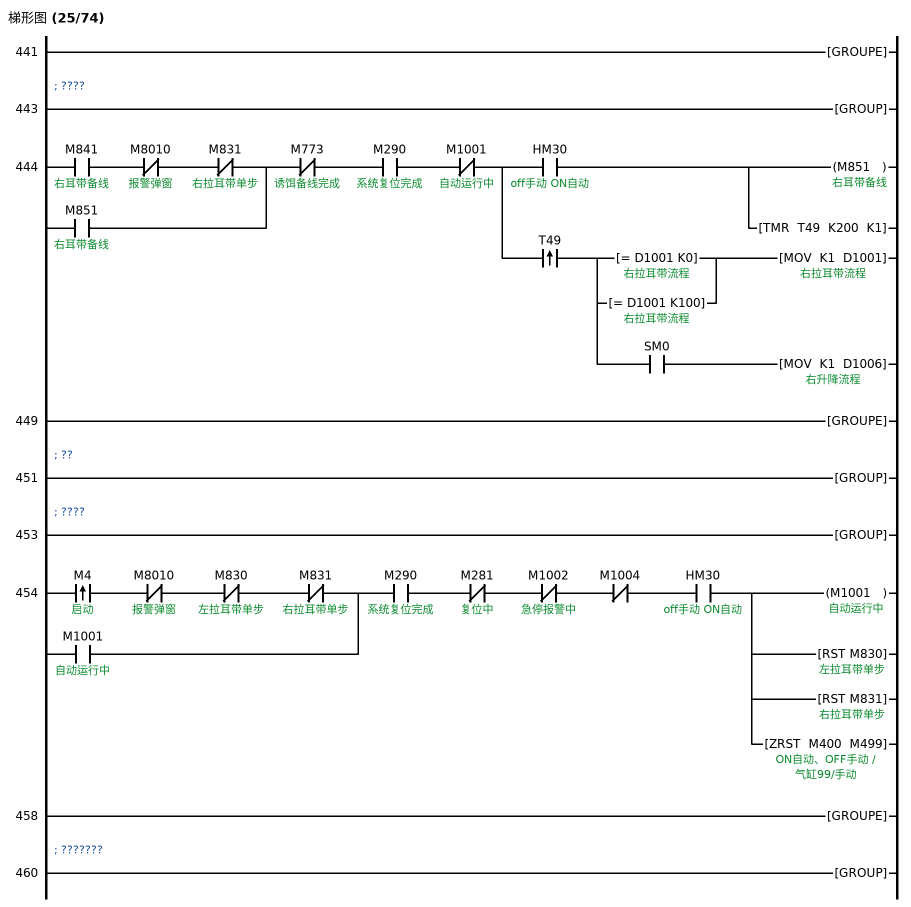
[picture p24: 梯形图 rows 441-460]
GROUPE
; ????
GROUP
LD     M841	; 右耳带备线
ANI    M8010	; 报警弹窗
ANI    M831	; 右拉耳带单步
OR     M851	; 右耳带备线
ANI    M773	; 诱饵备线完成
AND    M290	; 系统复位完成
ANI    M1001	; 自动运行中
MPS
AND    HM30	; off手动 ON自动
OUT    M851	; 右耳带备线
TMR    T49 K200 K1
MPP
ANDP   T49
MPS
LD=    D1001 K0	; 右拉耳带流程
OR=    D1001 K100	; 右拉耳带流程
ANB
MOV    K1 D1001	; 右拉耳带流程
MPP
AND    SM0
MOV    K1 D1006	; 右升降流程
GROUPE
; ??
GROUP
; ????
GROUP
LDP    M4	; 启动
ANI    M8010	; 报警弹窗
ANI    M830	; 左拉耳带单步
ANI    M831	; 右拉耳带单步
OR     M1001	; 自动运行中
AND    M290	; 系统复位完成
ANI    M281	; 复位中
ANI    M1002	; 急停报警中
ANI    M1004
AND    HM30	; off手动 ON自动
OUT    M1001	; 自动运行中
RST    M830	; 左拉耳带单步
RST    M831	; 右拉耳带单步
ZRST   M400 M499	; ON自动、OFF手动 / 气缸99/手动
GROUPE
; ???????
GROUP

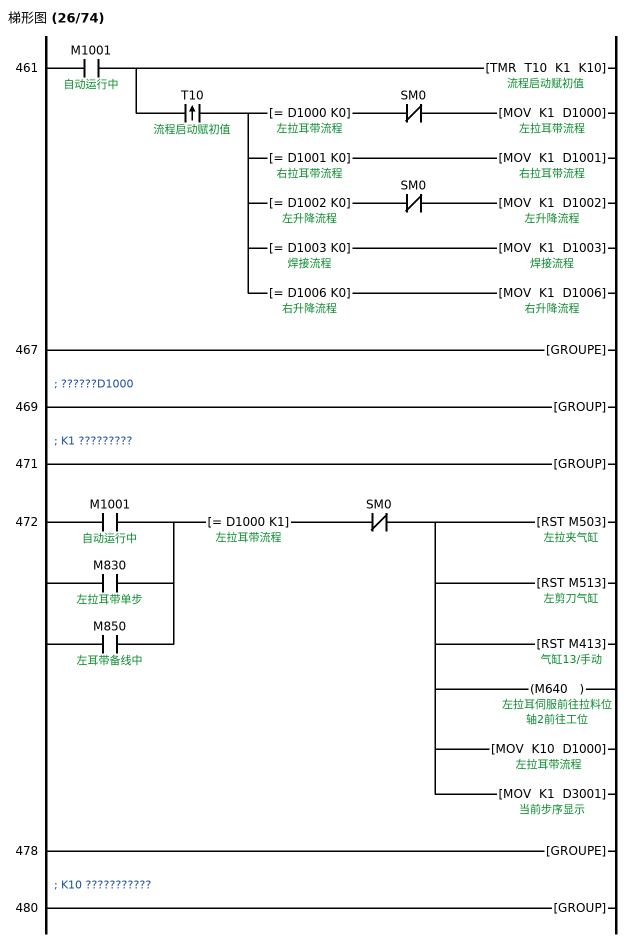
LD     M1001	; 自动运行中
TMR    T10 K1 K10	; 流程启动赋初值
ANDP   T10	; 流程启动赋初值
MPS
AND=   D1000 K0	; 左拉耳带流程
ANI    SM0
MOV    K1 D1000	; 左拉耳带流程
MRD
AND=   D1001 K0	; 右拉耳带流程
MOV    K1 D1001	; 右拉耳带流程
MRD
AND=   D1002 K0	; 左升降流程
ANI    SM0
MOV    K1 D1002	; 左升降流程
MRD
AND=   D1003 K0	; 焊接流程
MOV    K1 D1003	; 焊接流程
MPP
AND=   D1006 K0	; 右升降流程
MOV    K1 D1006	; 右升降流程
GROUPE
; ??????D1000
GROUP
; K1 ?????????
GROUP
LD     M1001	; 自动运行中
OR     M830	; 左拉耳带单步
OR     M850	; 左耳带备线中
AND=   D1000 K1	; 左拉耳带流程
ANI    SM0
RST    M503	; 左拉夹气缸
RST    M513	; 左剪刀气缸
RST    M413	; 气缸13/手动
OUT    M640	; 左拉耳伺服前往拉料位 轴2前往工位
MOV    K10 D1000	; 左拉耳带流程
MOV    K1 D3001	; 当前步序显示
GROUPE
; K10 ???????????
GROUP

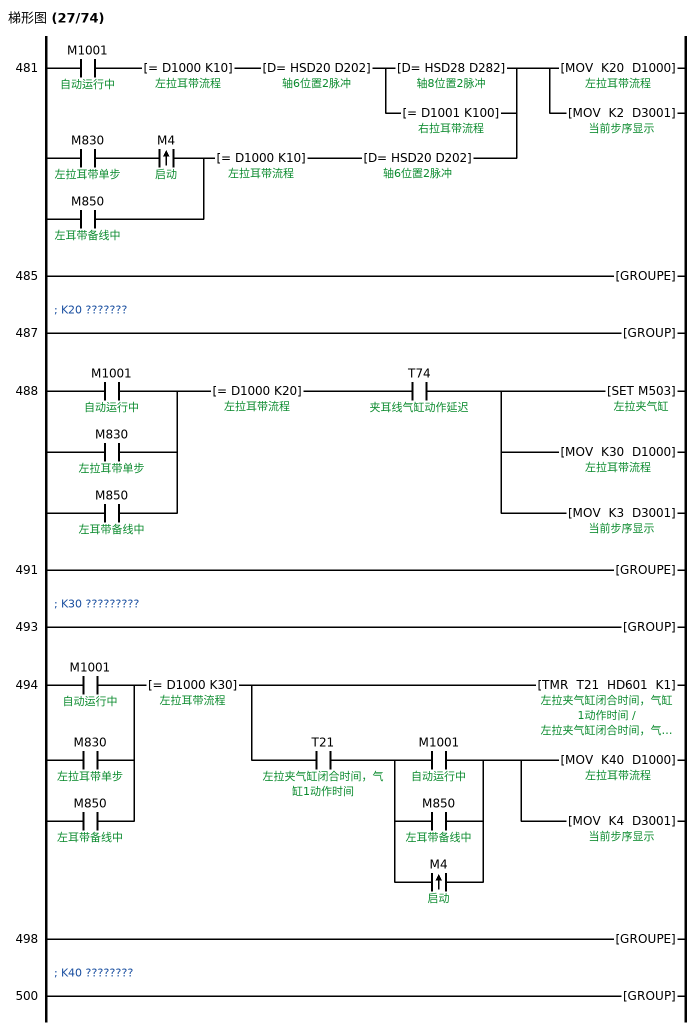
LD     M1001	; 自动运行中
AND=   D1000 K10	; 左拉耳带流程
DAND=  HSD20 D202	; 轴6位置2脉冲
DLD=   HSD28 D282	; 轴8位置2脉冲
OR=    D1001 K100	; 右拉耳带流程
ANB
LD     M830	; 左拉耳带单步
ANDP   M4	; 启动
OR     M850	; 左耳带备线中
AND=   D1000 K10	; 左拉耳带流程
DAND=  HSD20 D202	; 轴6位置2脉冲
ORB
MOV    K20 D1000	; 左拉耳带流程
MOV    K2 D3001	; 当前步序显示
GROUPE
; K20 ???????
GROUP
LD     M1001	; 自动运行中
OR     M830	; 左拉耳带单步
OR     M850	; 左耳带备线中
AND=   D1000 K20	; 左拉耳带流程
AND    T74	; 夹耳线气缸动作延迟
SET    M503	; 左拉夹气缸
MOV    K30 D1000	; 左拉耳带流程
MOV    K3 D3001	; 当前步序显示
GROUPE
; K30 ?????????
GROUP
LD     M1001	; 自动运行中
OR     M830	; 左拉耳带单步
OR     M850	; 左耳带备线中
AND=   D1000 K30	; 左拉耳带流程
TMR    T21 HD601 K1	; 左拉夹气缸闭合时间，气缸1动作时间 / 左拉夹气缸闭合时间，气缸1动作时间
AND    T21	; 左拉夹气缸闭合时间，气缸1动作时间
LD     M1001	; 自动运行中
OR     M850	; 左耳带备线中
ORP    M4	; 启动
ANB
MOV    K40 D1000	; 左拉耳带流程
MOV    K4 D3001	; 当前步序显示
GROUPE
; K40 ????????
GROUP

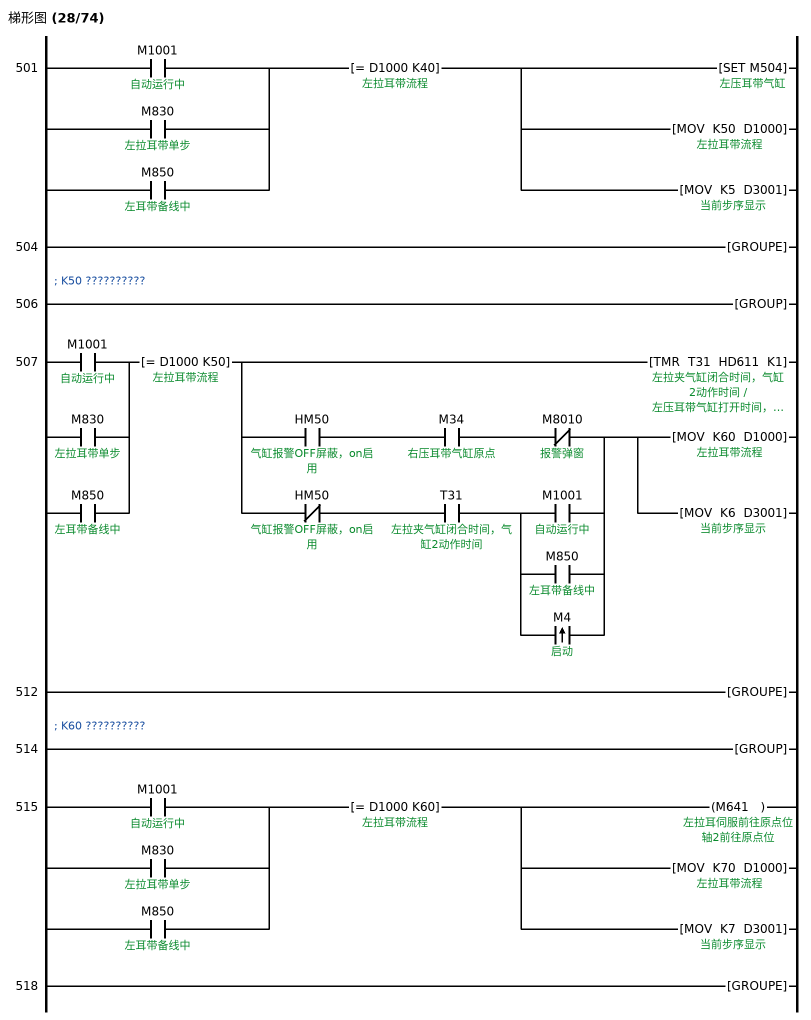
LD     M1001	; 自动运行中
OR     M830	; 左拉耳带单步
OR     M850	; 左耳带备线中
AND=   D1000 K40	; 左拉耳带流程
SET    M504	; 左压耳带气缸
MOV    K50 D1000	; 左拉耳带流程
MOV    K5 D3001	; 当前步序显示
GROUPE
; K50 ??????????
GROUP
LD     M1001	; 自动运行中
OR     M830	; 左拉耳带单步
OR     M850	; 左耳带备线中
AND=   D1000 K50	; 左拉耳带流程
TMR    T31 HD611 K1	; 左拉夹气缸闭合时间，气缸2动作时间 / 左压耳带气缸打开时间，气缸2动作时间
LD     HM50	; 气缸报警OFF屏蔽，on启用
AND    M34	; 右压耳带气缸原点
ANI    M8010	; 报警弹窗
LDI    HM50	; 气缸报警OFF屏蔽，on启用
AND    T31	; 左拉夹气缸闭合时间，气缸2动作时间
LD     M1001	; 自动运行中
OR     M850	; 左耳带备线中
ORP    M4	; 启动
ANB
ORB
ANB
MOV    K60 D1000	; 左拉耳带流程
MOV    K6 D3001	; 当前步序显示
GROUPE
; K60 ??????????
GROUP
LD     M1001	; 自动运行中
OR     M830	; 左拉耳带单步
OR     M850	; 左耳带备线中
AND=   D1000 K60	; 左拉耳带流程
OUT    M641	; 左拉耳伺服前往原点位 轴2前往原点位
MOV    K70 D1000	; 左拉耳带流程
MOV    K7 D3001	; 当前步序显示
GROUPE

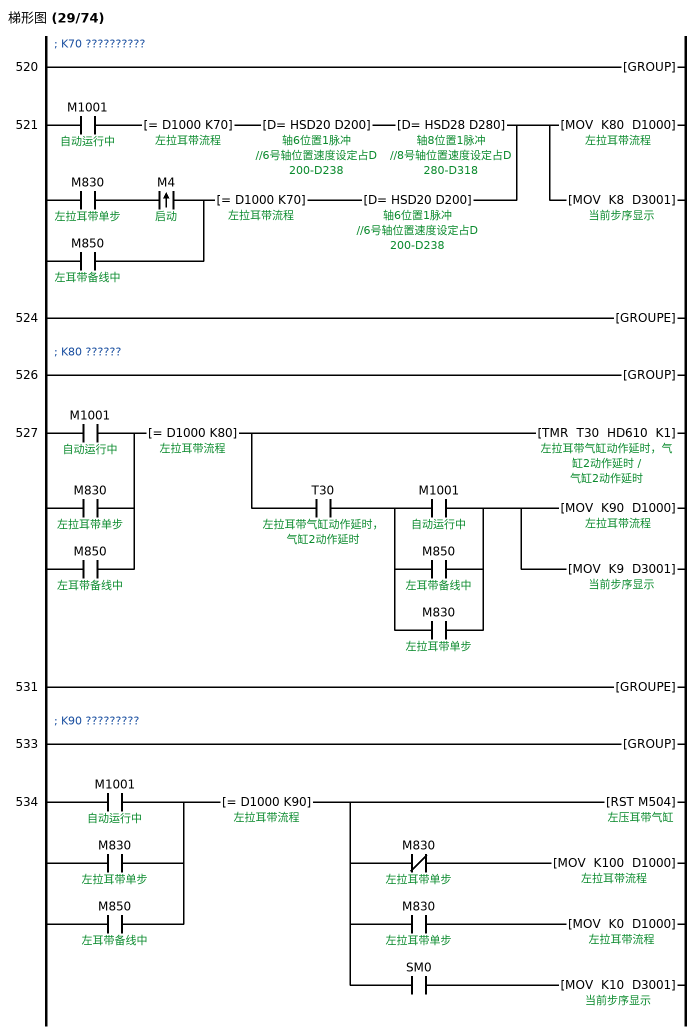
; K70 ??????????
GROUP
LD     M1001	; 自动运行中
AND=   D1000 K70	; 左拉耳带流程
DAND=  HSD20 D200	; 轴6位置1脉冲   //6号轴位置速度设定占D200-D238
DAND=  HSD28 D280	; 轴8位置1脉冲   //8号轴位置速度设定占D280-D318
LD     M830	; 左拉耳带单步
ANDP   M4	; 启动
OR     M850	; 左耳带备线中
AND=   D1000 K70	; 左拉耳带流程
DAND=  HSD20 D200	; 轴6位置1脉冲   //6号轴位置速度设定占D200-D238
ORB
MOV    K80 D1000	; 左拉耳带流程
MOV    K8 D3001	; 当前步序显示
GROUPE
; K80 ??????
GROUP
LD     M1001	; 自动运行中
OR     M830	; 左拉耳带单步
OR     M850	; 左耳带备线中
AND=   D1000 K80	; 左拉耳带流程
TMR    T30 HD610 K1	; 左拉耳带气缸动作延时，气缸2动作延时 / 气缸2动作延时
AND    T30	; 左拉耳带气缸动作延时，气缸2动作延时
LD     M1001	; 自动运行中
OR     M850	; 左耳带备线中
OR     M830	; 左拉耳带单步
ANB
MOV    K90 D1000	; 左拉耳带流程
MOV    K9 D3001	; 当前步序显示
GROUPE
; K90 ?????????
GROUP
LD     M1001	; 自动运行中
OR     M830	; 左拉耳带单步
OR     M850	; 左耳带备线中
AND=   D1000 K90	; 左拉耳带流程
RST    M504	; 左压耳带气缸
MPS
ANI    M830	; 左拉耳带单步
MOV    K100 D1000	; 左拉耳带流程
MRD
AND    M830	; 左拉耳带单步
MOV    K0 D1000	; 左拉耳带流程
MPP
AND    SM0
MOV    K10 D3001	; 当前步序显示

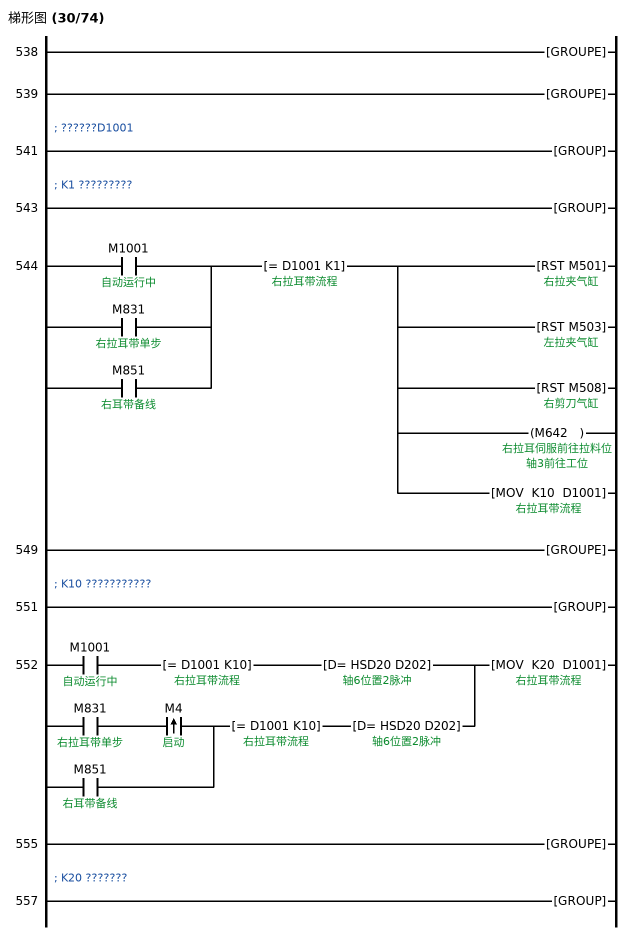
GROUPE
GROUPE
; ??????D1001
GROUP
; K1 ?????????
GROUP
LD     M1001	; 自动运行中
OR     M831	; 右拉耳带单步
OR     M851	; 右耳带备线
AND=   D1001 K1	; 右拉耳带流程
RST    M501	; 右拉夹气缸
RST    M503	; 左拉夹气缸
RST    M508	; 右剪刀气缸
OUT    M642	; 右拉耳伺服前往拉料位 轴3前往工位
MOV    K10 D1001	; 右拉耳带流程
GROUPE
; K10 ???????????
GROUP
LD     M1001	; 自动运行中
AND=   D1001 K10	; 右拉耳带流程
DAND=  HSD20 D202	; 轴6位置2脉冲
LD     M831	; 右拉耳带单步
ANDP   M4	; 启动
OR     M851	; 右耳带备线
AND=   D1001 K10	; 右拉耳带流程
DAND=  HSD20 D202	; 轴6位置2脉冲
ORB
MOV    K20 D1001	; 右拉耳带流程
GROUPE
; K20 ???????
GROUP

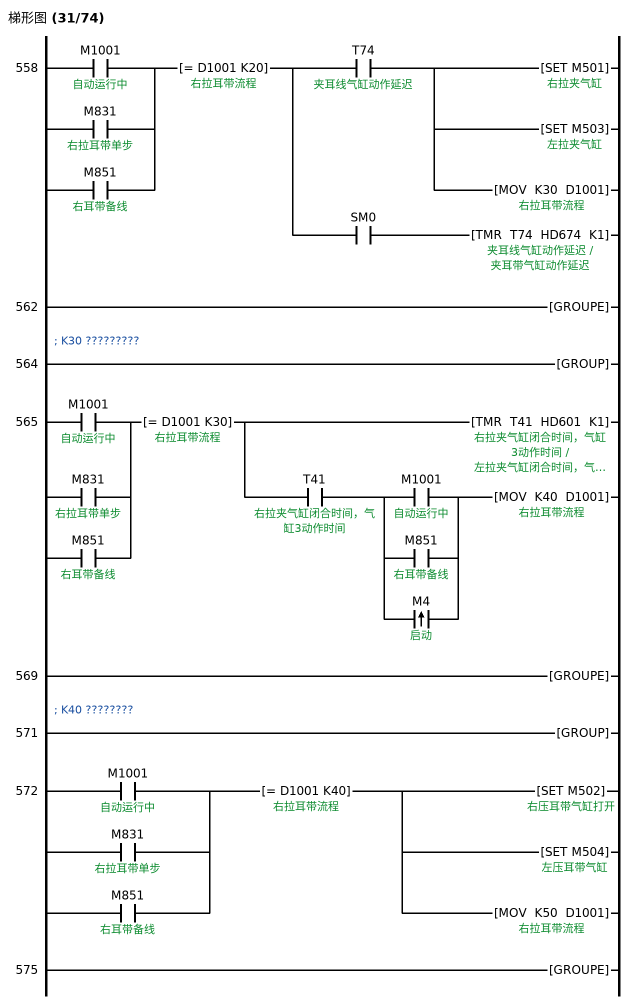
LD     M1001	; 自动运行中
OR     M831	; 右拉耳带单步
OR     M851	; 右耳带备线
AND=   D1001 K20	; 右拉耳带流程
MPS
AND    T74	; 夹耳线气缸动作延迟
SET    M501	; 右拉夹气缸
SET    M503	; 左拉夹气缸
MOV    K30 D1001	; 右拉耳带流程
MPP
AND    SM0
TMR    T74 HD674 K1	; 夹耳线气缸动作延迟 / 夹耳带气缸动作延迟
GROUPE
; K30 ?????????
GROUP
LD     M1001	; 自动运行中
OR     M831	; 右拉耳带单步
OR     M851	; 右耳带备线
AND=   D1001 K30	; 右拉耳带流程
TMR    T41 HD601 K1	; 右拉夹气缸闭合时间，气缸3动作时间 / 左拉夹气缸闭合时间，气缸1动作时间
AND    T41	; 右拉夹气缸闭合时间，气缸3动作时间
LD     M1001	; 自动运行中
OR     M851	; 右耳带备线
ORP    M4	; 启动
ANB
MOV    K40 D1001	; 右拉耳带流程
GROUPE
; K40 ????????
GROUP
LD     M1001	; 自动运行中
OR     M831	; 右拉耳带单步
OR     M851	; 右耳带备线
AND=   D1001 K40	; 右拉耳带流程
SET    M502	; 右压耳带气缸打开
SET    M504	; 左压耳带气缸
MOV    K50 D1001	; 右拉耳带流程
GROUPE

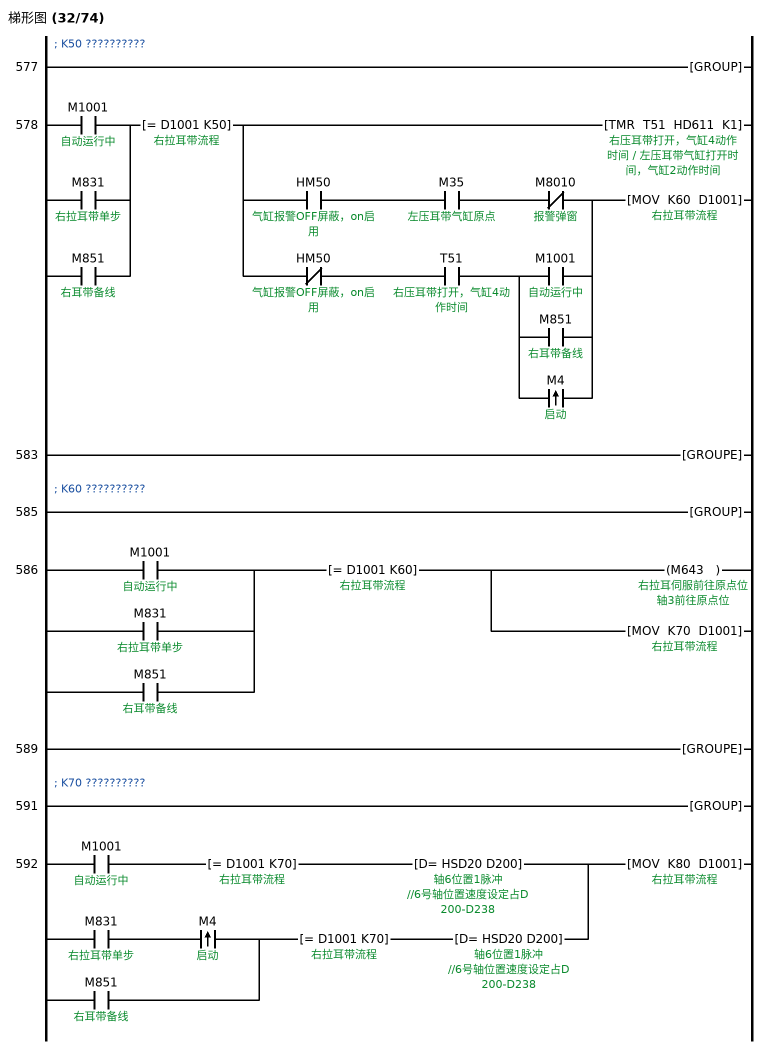
; K50 ??????????
GROUP
LD     M1001	; 自动运行中
OR     M831	; 右拉耳带单步
OR     M851	; 右耳带备线
AND=   D1001 K50	; 右拉耳带流程
TMR    T51 HD611 K1	; 右压耳带打开，气缸4动作时间 / 左压耳带气缸打开时间，气缸2动作时间
LD     HM50	; 气缸报警OFF屏蔽，on启用
AND    M35	; 左压耳带气缸原点
ANI    M8010	; 报警弹窗
LDI    HM50	; 气缸报警OFF屏蔽，on启用
AND    T51	; 右压耳带打开，气缸4动作时间
LD     M1001	; 自动运行中
OR     M851	; 右耳带备线
ORP    M4	; 启动
ANB
ORB
ANB
MOV    K60 D1001	; 右拉耳带流程
GROUPE
; K60 ??????????
GROUP
LD     M1001	; 自动运行中
OR     M831	; 右拉耳带单步
OR     M851	; 右耳带备线
AND=   D1001 K60	; 右拉耳带流程
OUT    M643	; 右拉耳伺服前往原点位 轴3前往原点位
MOV    K70 D1001	; 右拉耳带流程
GROUPE
; K70 ??????????
GROUP
LD     M1001	; 自动运行中
AND=   D1001 K70	; 右拉耳带流程
DAND=  HSD20 D200	; 轴6位置1脉冲   //6号轴位置速度设定占D200-D238
LD     M831	; 右拉耳带单步
ANDP   M4	; 启动
OR     M851	; 右耳带备线
AND=   D1001 K70	; 右拉耳带流程
DAND=  HSD20 D200	; 轴6位置1脉冲   //6号轴位置速度设定占D200-D238
ORB
MOV    K80 D1001	; 右拉耳带流程

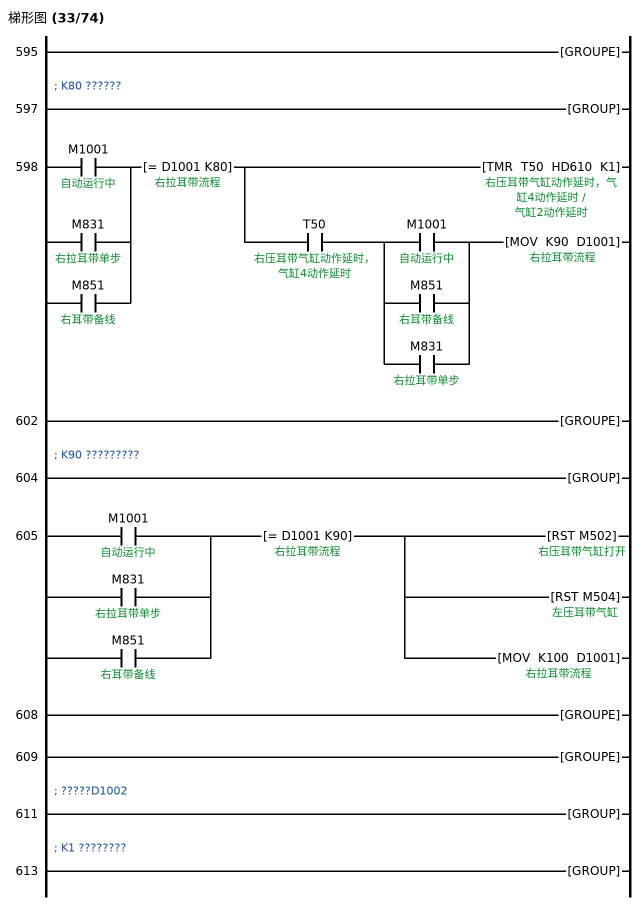
GROUPE
; K80 ??????
GROUP
LD     M1001	; 自动运行中
OR     M831	; 右拉耳带单步
OR     M851	; 右耳带备线
AND=   D1001 K80	; 右拉耳带流程
TMR    T50 HD610 K1	; 右压耳带气缸动作延时，气缸4动作延时 / 气缸2动作延时
AND    T50	; 右压耳带气缸动作延时，气缸4动作延时
LD     M1001	; 自动运行中
OR     M851	; 右耳带备线
OR     M831	; 右拉耳带单步
ANB
MOV    K90 D1001	; 右拉耳带流程
GROUPE
; K90 ?????????
GROUP
LD     M1001	; 自动运行中
OR     M831	; 右拉耳带单步
OR     M851	; 右耳带备线
AND=   D1001 K90	; 右拉耳带流程
RST    M502	; 右压耳带气缸打开
RST    M504	; 左压耳带气缸
MOV    K100 D1001	; 右拉耳带流程
GROUPE
GROUPE
; ?????D1002
GROUP
; K1 ????????
GROUP

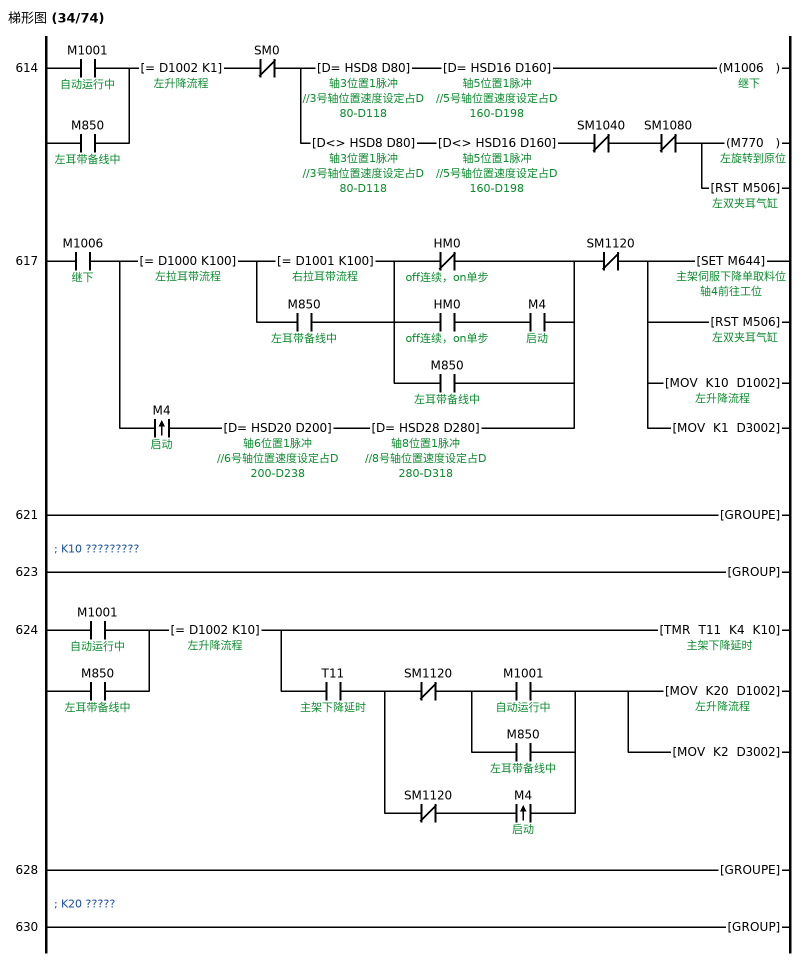
LD     M1001	; 自动运行中
OR     M850	; 左耳带备线中
AND=   D1002 K1	; 左升降流程
ANI    SM0
MPS
DAND=  HSD8 D80	; 轴3位置1脉冲   //3号轴位置速度设定占D80-D118
DAND=  HSD16 D160	; 轴5位置1脉冲   //5号轴位置速度设定占D160-D198
OUT    M1006	; 继下
MPP
DAND<> HSD8 D80	; 轴3位置1脉冲   //3号轴位置速度设定占D80-D118
DAND<> HSD16 D160	; 轴5位置1脉冲   //5号轴位置速度设定占D160-D198
ANI    SM1040
ANI    SM1080
OUT    M770	; 左旋转到原位
RST    M506	; 左双夹耳气缸
LD     M1006	; 继下
LD=    D1000 K100	; 左拉耳带流程
LD=    D1001 K100	; 右拉耳带流程
OR     M850	; 左耳带备线中
ANB
LDI    HM0	; off连续，on单步
LD     HM0	; off连续，on单步
AND    M4	; 启动
ORB
OR     M850	; 左耳带备线中
ANB
LDP    M4	; 启动
DAND=  HSD20 D200	; 轴6位置1脉冲   //6号轴位置速度设定占D200-D238
DAND=  HSD28 D280	; 轴8位置1脉冲   //8号轴位置速度设定占D280-D318
ORB
ANB
ANI    SM1120
SET    M644	; 主架伺服下降单取料位 轴4前往工位
RST    M506	; 左双夹耳气缸
MOV    K10 D1002	; 左升降流程
MOV    K1 D3002
GROUPE
; K10 ?????????
GROUP
LD     M1001	; 自动运行中
OR     M850	; 左耳带备线中
AND=   D1002 K10	; 左升降流程
TMR    T11 K4 K10	; 主架下降延时
AND    T11	; 主架下降延时
LDI    SM1120
LD     M1001	; 自动运行中
OR     M850	; 左耳带备线中
ANB
LDI    SM1120
ANDP   M4	; 启动
ORB
ANB
MOV    K20 D1002	; 左升降流程
MOV    K2 D3002
GROUPE
; K20 ?????
GROUP

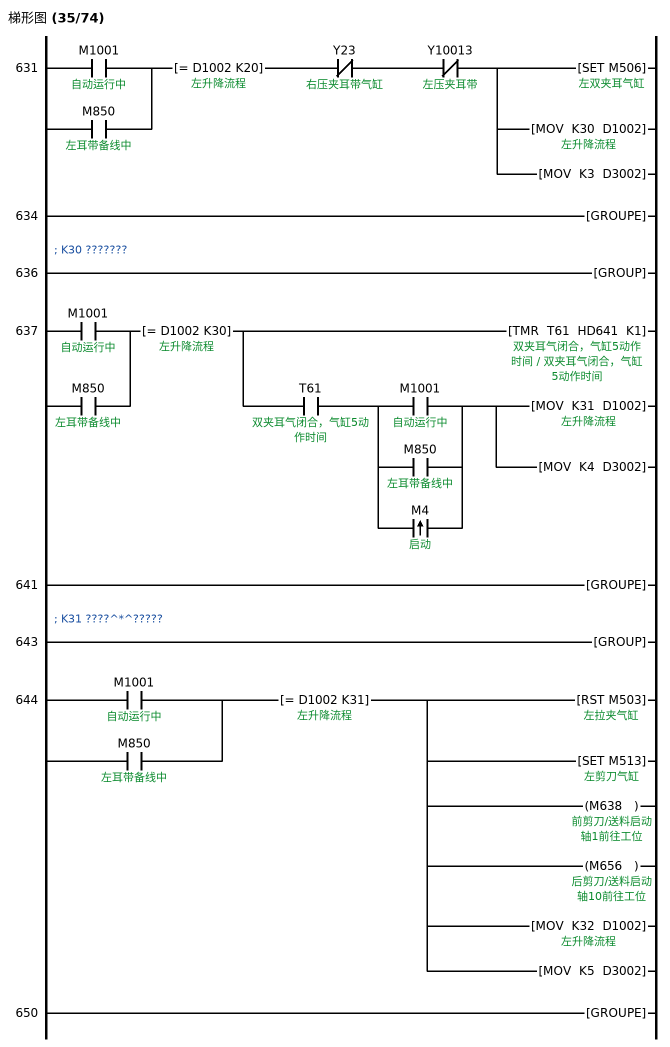
LD     M1001	; 自动运行中
OR     M850	; 左耳带备线中
AND=   D1002 K20	; 左升降流程
ANI    Y23	; 右压夹耳带气缸
ANI    Y10013	; 左压夹耳带
SET    M506	; 左双夹耳气缸
MOV    K30 D1002	; 左升降流程
MOV    K3 D3002
GROUPE
; K30 ???????
GROUP
LD     M1001	; 自动运行中
OR     M850	; 左耳带备线中
AND=   D1002 K30	; 左升降流程
TMR    T61 HD641 K1	; 双夹耳气闭合，气缸5动作时间 / 双夹耳气闭合，气缸5动作时间
AND    T61	; 双夹耳气闭合，气缸5动作时间
LD     M1001	; 自动运行中
OR     M850	; 左耳带备线中
ORP    M4	; 启动
ANB
MOV    K31 D1002	; 左升降流程
MOV    K4 D3002
GROUPE
; K31 ????^*^?????
GROUP
LD     M1001	; 自动运行中
OR     M850	; 左耳带备线中
AND=   D1002 K31	; 左升降流程
RST    M503	; 左拉夹气缸
SET    M513	; 左剪刀气缸
OUT    M638	; 前剪刀/送料启动 轴1前往工位
OUT    M656	; 后剪刀/送料启动 轴10前往工位
MOV    K32 D1002	; 左升降流程
MOV    K5 D3002
GROUPE

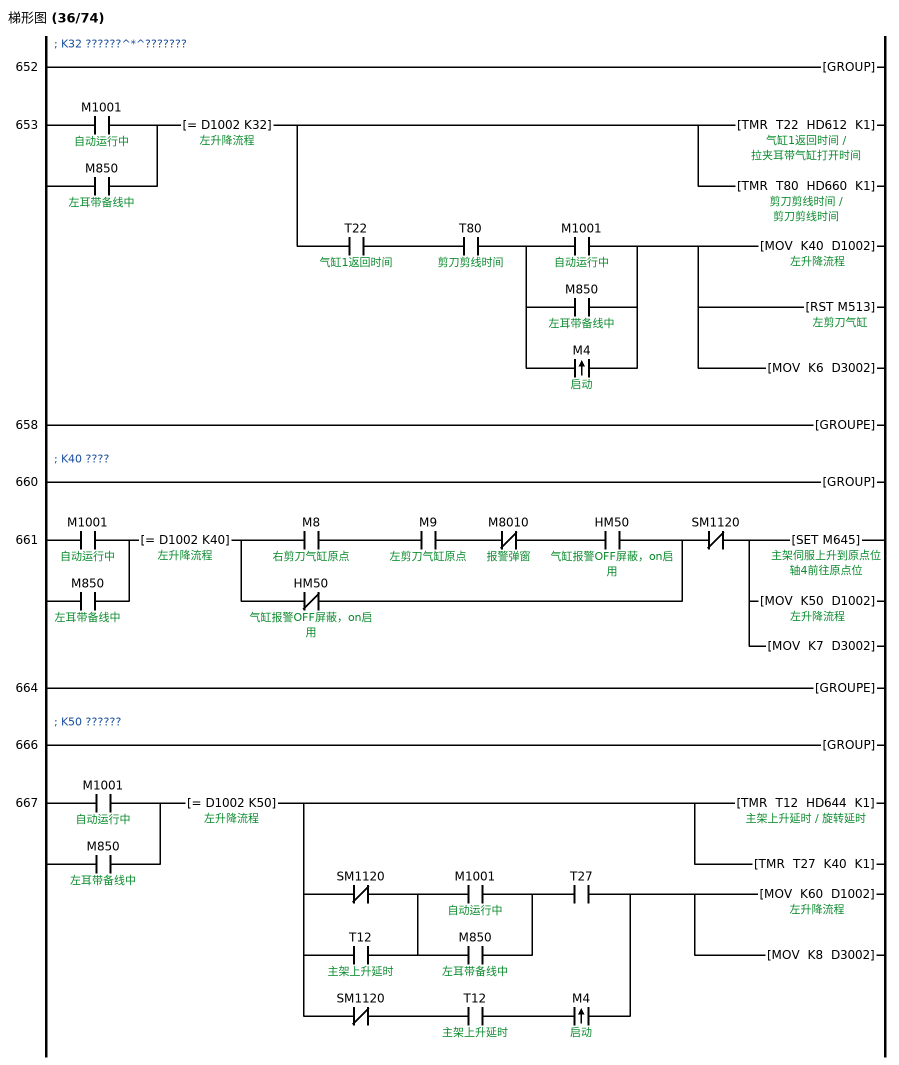
; K32 ??????^*^???????
GROUP
LD     M1001	; 自动运行中
OR     M850	; 左耳带备线中
AND=   D1002 K32	; 左升降流程
TMR    T22 HD612 K1	; 气缸1返回时间 / 拉夹耳带气缸打开时间
TMR    T80 HD660 K1	; 剪刀剪线时间 / 剪刀剪线时间
AND    T22	; 气缸1返回时间
AND    T80	; 剪刀剪线时间
LD     M1001	; 自动运行中
OR     M850	; 左耳带备线中
ORP    M4	; 启动
ANB
MOV    K40 D1002	; 左升降流程
RST    M513	; 左剪刀气缸
MOV    K6 D3002
GROUPE
; K40 ????
GROUP
LD     M1001	; 自动运行中
OR     M850	; 左耳带备线中
AND=   D1002 K40	; 左升降流程
LD     M8	; 右剪刀气缸原点
AND    M9	; 左剪刀气缸原点
ANI    M8010	; 报警弹窗
AND    HM50	; 气缸报警OFF屏蔽，on启用
ORI    HM50	; 气缸报警OFF屏蔽，on启用
ANB
ANI    SM1120
SET    M645	; 主架伺服上升到原点位 轴4前往原点位
MOV    K50 D1002	; 左升降流程
MOV    K7 D3002
GROUPE
; K50 ??????
GROUP
LD     M1001	; 自动运行中
OR     M850	; 左耳带备线中
AND=   D1002 K50	; 左升降流程
TMR    T12 HD644 K1	; 主架上升延时 / 旋转延时
TMR    T27 K40 K1
LDI    SM1120
OR     T12	; 主架上升延时
LD     M1001	; 自动运行中
OR     M850	; 左耳带备线中
ANB
AND    T27
LDI    SM1120
AND    T12	; 主架上升延时
ANDP   M4	; 启动
ORB
ANB
MOV    K60 D1002	; 左升降流程
MOV    K8 D3002

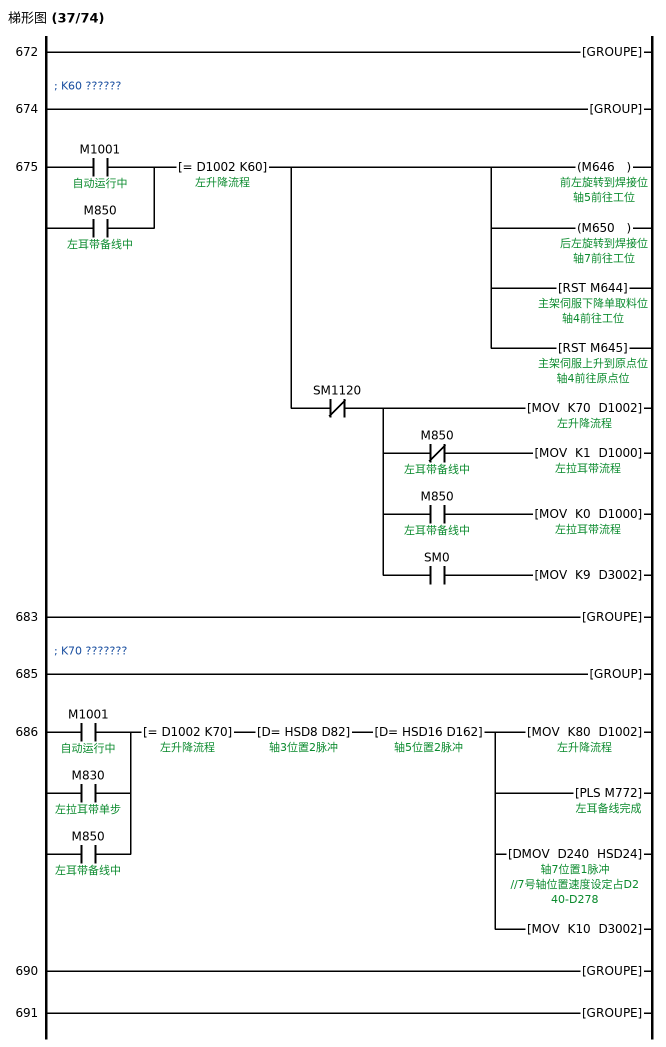
GROUPE
; K60 ??????
GROUP
LD     M1001	; 自动运行中
OR     M850	; 左耳带备线中
AND=   D1002 K60	; 左升降流程
OUT    M646	; 前左旋转到焊接位 轴5前往工位
OUT    M650	; 后左旋转到焊接位 轴7前往工位
RST    M644	; 主架伺服下降单取料位 轴4前往工位
RST    M645	; 主架伺服上升到原点位 轴4前往原点位
ANI    SM1120
MOV    K70 D1002	; 左升降流程
MPS
ANI    M850	; 左耳带备线中
MOV    K1 D1000	; 左拉耳带流程
MRD
AND    M850	; 左耳带备线中
MOV    K0 D1000	; 左拉耳带流程
MPP
AND    SM0
MOV    K9 D3002
GROUPE
; K70 ???????
GROUP
LD     M1001	; 自动运行中
OR     M830	; 左拉耳带单步
OR     M850	; 左耳带备线中
AND=   D1002 K70	; 左升降流程
DAND=  HSD8 D82	; 轴3位置2脉冲
DAND=  HSD16 D162	; 轴5位置2脉冲
MOV    K80 D1002	; 左升降流程
PLS    M772	; 左耳备线完成
DMOV   D240 HSD24	; 轴7位置1脉冲   //7号轴位置速度设定占D240-D278
MOV    K10 D3002
GROUPE
GROUPE

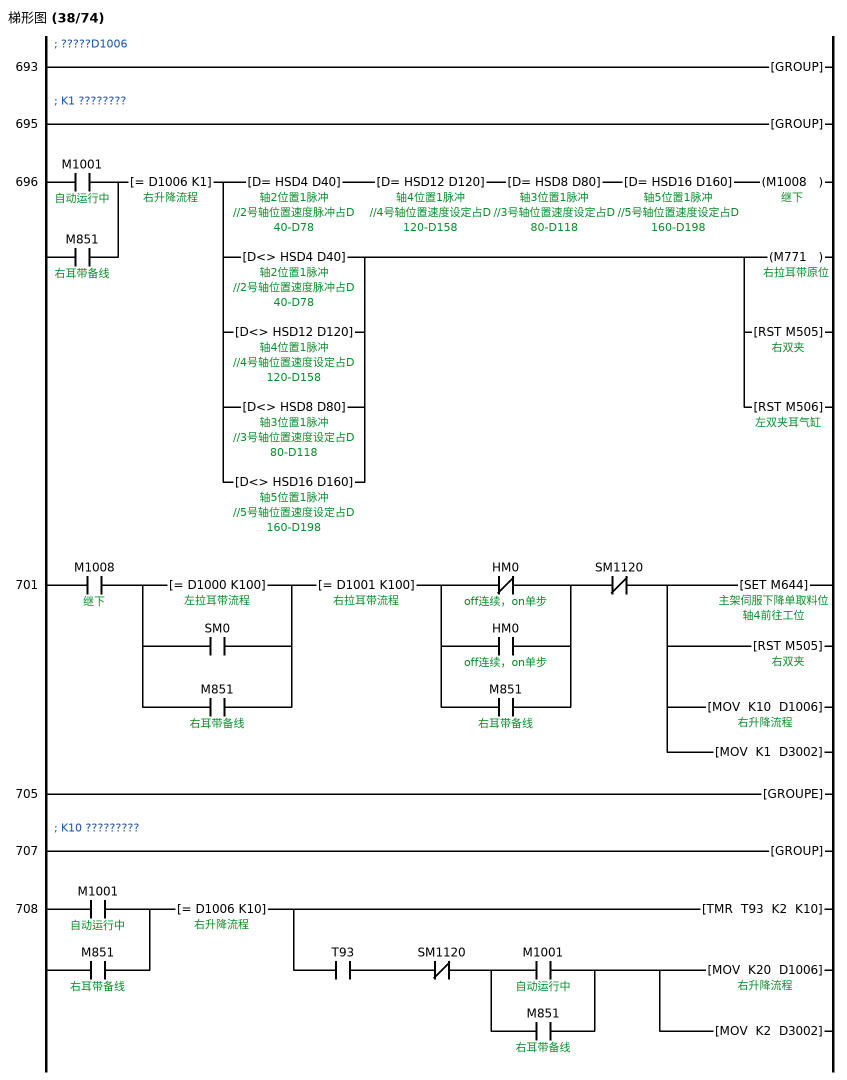
; ?????D1006
GROUP
; K1 ????????
GROUP
LD     M1001	; 自动运行中
OR     M851	; 右耳带备线
AND=   D1006 K1	; 右升降流程
MPS
DAND=  HSD4 D40	; 轴2位置1脉冲    //2号轴位置速度脉冲占D40-D78
DAND=  HSD12 D120	; 轴4位置1脉冲   //4号轴位置速度设定占D120-D158
DAND=  HSD8 D80	; 轴3位置1脉冲   //3号轴位置速度设定占D80-D118
DAND=  HSD16 D160	; 轴5位置1脉冲   //5号轴位置速度设定占D160-D198
OUT    M1008	; 继下
MPP
DLD<>  HSD4 D40	; 轴2位置1脉冲    //2号轴位置速度脉冲占D40-D78
DOR<>  HSD12 D120	; 轴4位置1脉冲   //4号轴位置速度设定占D120-D158
DOR<>  HSD8 D80	; 轴3位置1脉冲   //3号轴位置速度设定占D80-D118
DOR<>  HSD16 D160	; 轴5位置1脉冲   //5号轴位置速度设定占D160-D198
ANB
OUT    M771	; 右拉耳带原位
RST    M505	; 右双夹
RST    M506	; 左双夹耳气缸
LD     M1008	; 继下
LD=    D1000 K100	; 左拉耳带流程
OR     SM0
OR     M851	; 右耳带备线
ANB
AND=   D1001 K100	; 右拉耳带流程
LDI    HM0	; off连续，on单步
OR     HM0	; off连续，on单步
OR     M851	; 右耳带备线
ANB
ANI    SM1120
SET    M644	; 主架伺服下降单取料位 轴4前往工位
RST    M505	; 右双夹
MOV    K10 D1006	; 右升降流程
MOV    K1 D3002
GROUPE
; K10 ?????????
GROUP
LD     M1001	; 自动运行中
OR     M851	; 右耳带备线
AND=   D1006 K10	; 右升降流程
TMR    T93 K2 K10
AND    T93
ANI    SM1120
LD     M1001	; 自动运行中
OR     M851	; 右耳带备线
ANB
MOV    K20 D1006	; 右升降流程
MOV    K2 D3002

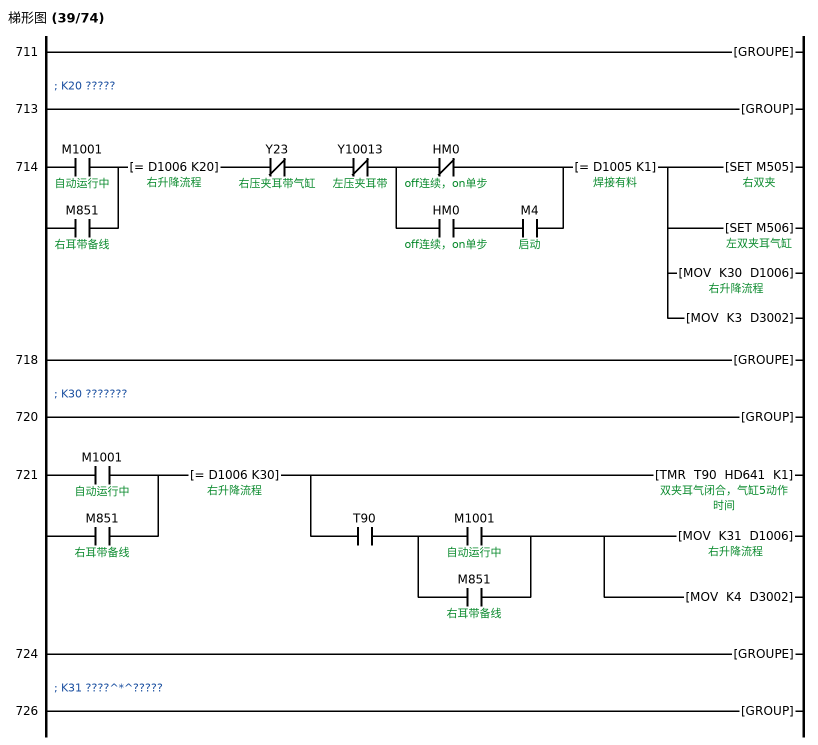
GROUPE
; K20 ?????
GROUP
LD     M1001	; 自动运行中
OR     M851	; 右耳带备线
AND=   D1006 K20	; 右升降流程
ANI    Y23	; 右压夹耳带气缸
ANI    Y10013	; 左压夹耳带
LDI    HM0	; off连续，on单步
LD     HM0	; off连续，on单步
AND    M4	; 启动
ORB
ANB
AND=   D1005 K1	; 焊接有料
SET    M505	; 右双夹
SET    M506	; 左双夹耳气缸
MOV    K30 D1006	; 右升降流程
MOV    K3 D3002
GROUPE
; K30 ???????
GROUP
LD     M1001	; 自动运行中
OR     M851	; 右耳带备线
AND=   D1006 K30	; 右升降流程
TMR    T90 HD641 K1	; 双夹耳气闭合，气缸5动作时间
AND    T90
LD     M1001	; 自动运行中
OR     M851	; 右耳带备线
ANB
MOV    K31 D1006	; 右升降流程
MOV    K4 D3002
GROUPE
; K31 ????^*^?????
GROUP

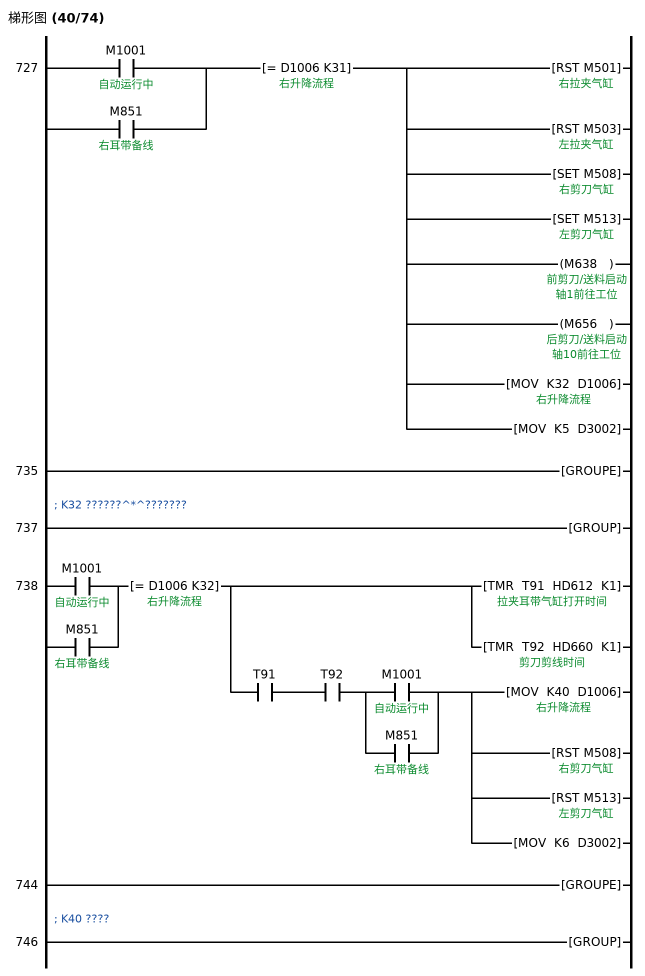
LD     M1001	; 自动运行中
OR     M851	; 右耳带备线
AND=   D1006 K31	; 右升降流程
RST    M501	; 右拉夹气缸
RST    M503	; 左拉夹气缸
SET    M508	; 右剪刀气缸
SET    M513	; 左剪刀气缸
OUT    M638	; 前剪刀/送料启动 轴1前往工位
OUT    M656	; 后剪刀/送料启动 轴10前往工位
MOV    K32 D1006	; 右升降流程
MOV    K5 D3002
GROUPE
; K32 ??????^*^???????
GROUP
LD     M1001	; 自动运行中
OR     M851	; 右耳带备线
AND=   D1006 K32	; 右升降流程
TMR    T91 HD612 K1	; 拉夹耳带气缸打开时间
TMR    T92 HD660 K1	; 剪刀剪线时间
AND    T91
AND    T92
LD     M1001	; 自动运行中
OR     M851	; 右耳带备线
ANB
MOV    K40 D1006	; 右升降流程
RST    M508	; 右剪刀气缸
RST    M513	; 左剪刀气缸
MOV    K6 D3002
GROUPE
; K40 ????
GROUP

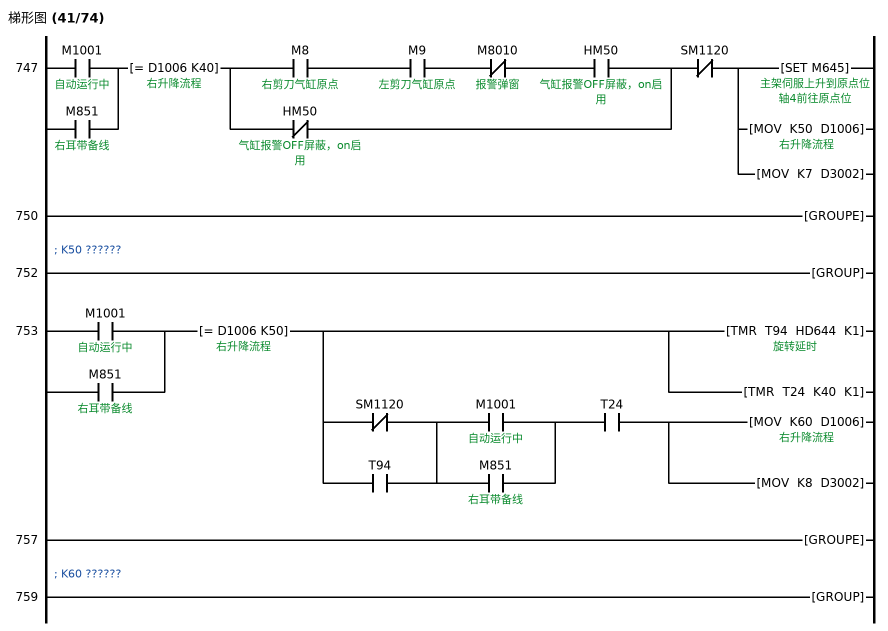
LD     M1001	; 自动运行中
OR     M851	; 右耳带备线
AND=   D1006 K40	; 右升降流程
LD     M8	; 右剪刀气缸原点
AND    M9	; 左剪刀气缸原点
ANI    M8010	; 报警弹窗
AND    HM50	; 气缸报警OFF屏蔽，on启用
ORI    HM50	; 气缸报警OFF屏蔽，on启用
ANB
ANI    SM1120
SET    M645	; 主架伺服上升到原点位 轴4前往原点位
MOV    K50 D1006	; 右升降流程
MOV    K7 D3002
GROUPE
; K50 ??????
GROUP
LD     M1001	; 自动运行中
OR     M851	; 右耳带备线
AND=   D1006 K50	; 右升降流程
TMR    T94 HD644 K1	; 旋转延时
TMR    T24 K40 K1
LDI    SM1120
OR     T94
ANB
LD     M1001	; 自动运行中
OR     M851	; 右耳带备线
ANB
AND    T24
MOV    K60 D1006	; 右升降流程
MOV    K8 D3002
GROUPE
; K60 ??????
GROUP

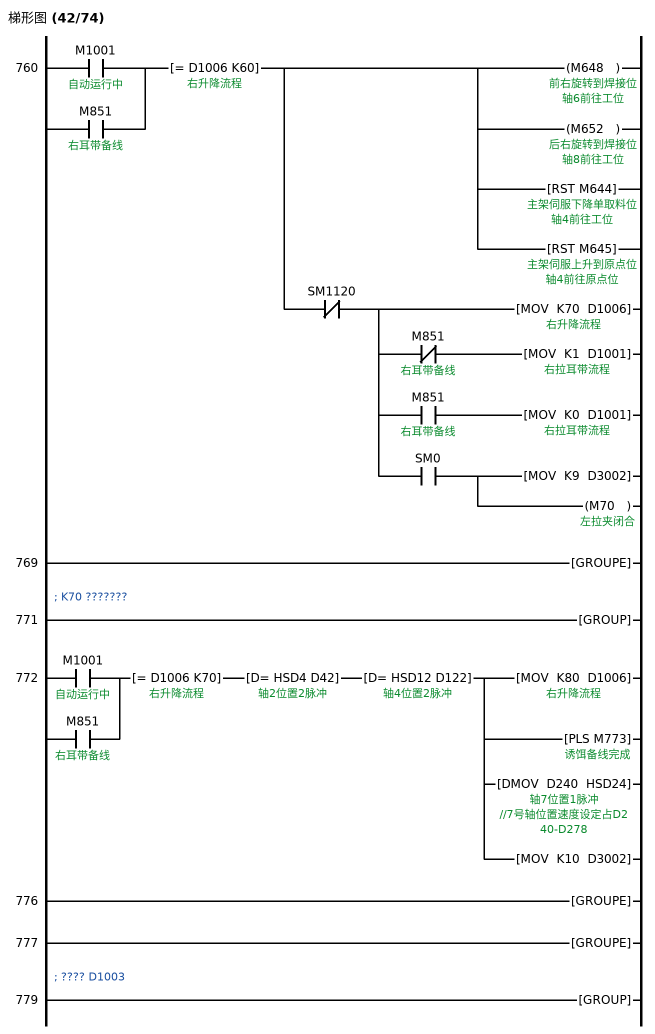
LD     M1001	; 自动运行中
OR     M851	; 右耳带备线
AND=   D1006 K60	; 右升降流程
OUT    M648	; 前右旋转到焊接位 轴6前往工位
OUT    M652	; 后右旋转到焊接位 轴8前往工位
RST    M644	; 主架伺服下降单取料位 轴4前往工位
RST    M645	; 主架伺服上升到原点位 轴4前往原点位
ANI    SM1120
MOV    K70 D1006	; 右升降流程
MPS
ANI    M851	; 右耳带备线
MOV    K1 D1001	; 右拉耳带流程
MRD
AND    M851	; 右耳带备线
MOV    K0 D1001	; 右拉耳带流程
MPP
AND    SM0
MOV    K9 D3002
OUT    M70	; 左拉夹闭合
GROUPE
; K70 ???????
GROUP
LD     M1001	; 自动运行中
OR     M851	; 右耳带备线
AND=   D1006 K70	; 右升降流程
DAND=  HSD4 D42	; 轴2位置2脉冲
DAND=  HSD12 D122	; 轴4位置2脉冲
MOV    K80 D1006	; 右升降流程
PLS    M773	; 诱饵备线完成
DMOV   D240 HSD24	; 轴7位置1脉冲   //7号轴位置速度设定占D240-D278
MOV    K10 D3002
GROUPE
GROUPE
; ???? D1003
GROUP

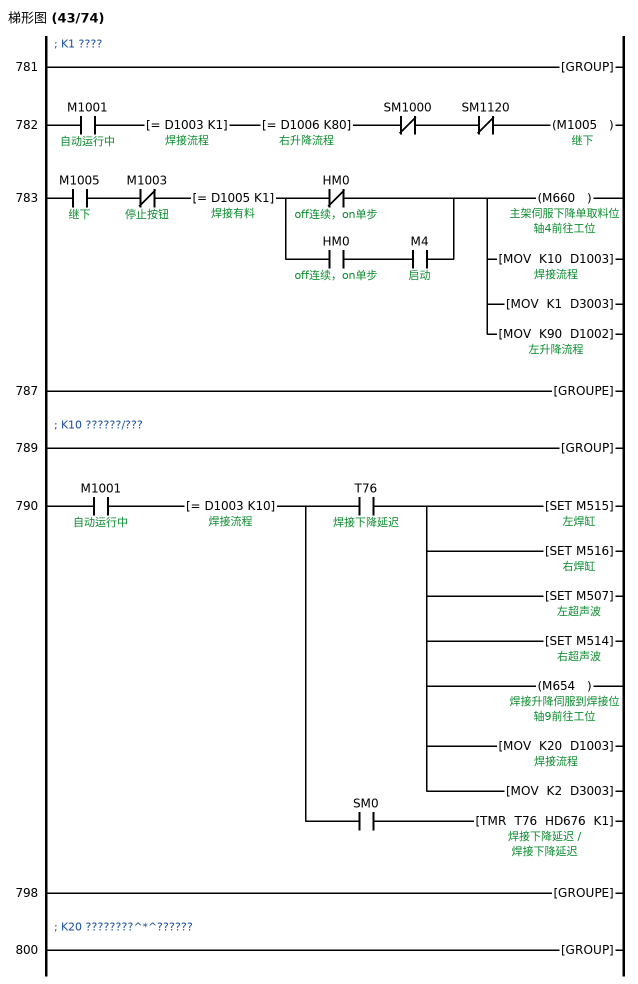
; K1 ????
GROUP
LD     M1001	; 自动运行中
AND=   D1003 K1	; 焊接流程
AND=   D1006 K80	; 右升降流程
ANI    SM1000
ANI    SM1120
OUT    M1005	; 继下
LD     M1005	; 继下
ANI    M1003	; 停止按钮
AND=   D1005 K1	; 焊接有料
LDI    HM0	; off连续，on单步
LD     HM0	; off连续，on单步
AND    M4	; 启动
ORB
ANB
OUT    M660	; 主架伺服下降单取料位 轴4前往工位
MOV    K10 D1003	; 焊接流程
MOV    K1 D3003
MOV    K90 D1002	; 左升降流程
GROUPE
; K10 ??????/???
GROUP
LD     M1001	; 自动运行中
AND=   D1003 K10	; 焊接流程
MPS
AND    T76	; 焊接下降延迟
SET    M515	; 左焊缸
SET    M516	; 右焊缸
SET    M507	; 左超声波
SET    M514	; 右超声波
OUT    M654	; 焊接升降伺服到焊接位 轴9前往工位
MOV    K20 D1003	; 焊接流程
MOV    K2 D3003
MPP
AND    SM0
TMR    T76 HD676 K1	; 焊接下降延迟 / 焊接下降延迟
GROUPE
; K20 ????????^*^??????
GROUP

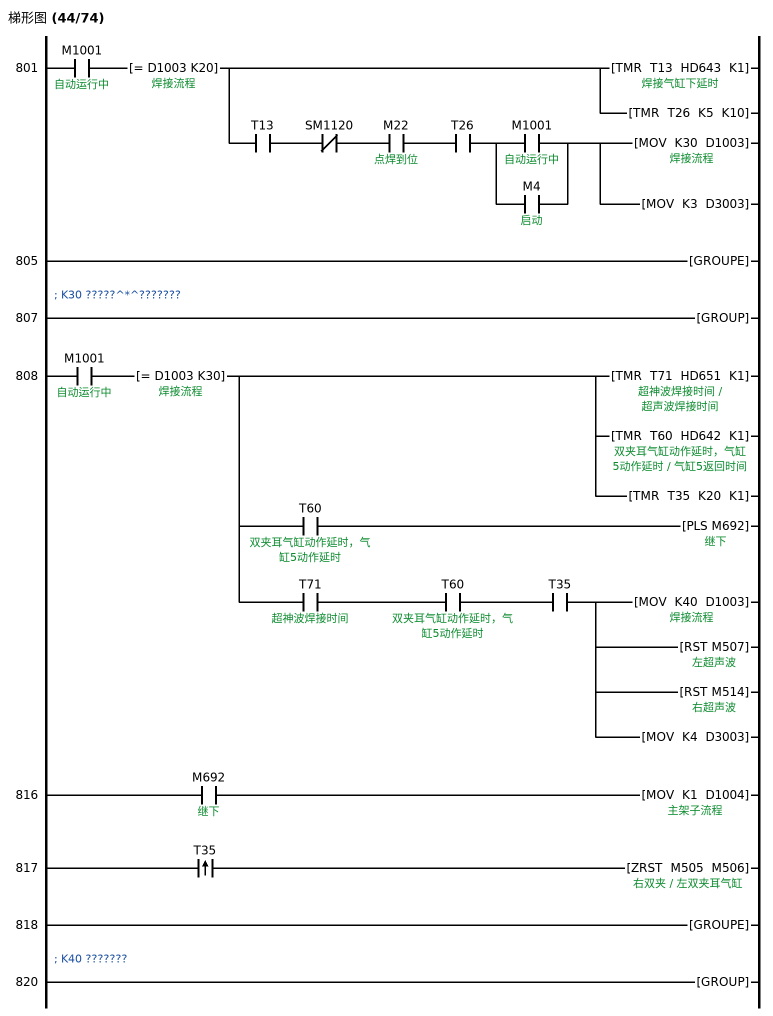
LD     M1001	; 自动运行中
AND=   D1003 K20	; 焊接流程
TMR    T13 HD643 K1	; 焊接气缸下延时
TMR    T26 K5 K10
AND    T13
ANI    SM1120
AND    M22	; 点焊到位
AND    T26
LD     M1001	; 自动运行中
OR     M4	; 启动
ANB
MOV    K30 D1003	; 焊接流程
MOV    K3 D3003
GROUPE
; K30 ?????^*^???????
GROUP
LD     M1001	; 自动运行中
AND=   D1003 K30	; 焊接流程
TMR    T71 HD651 K1	; 超神波焊接时间 / 超声波焊接时间
TMR    T60 HD642 K1	; 双夹耳气缸动作延时，气缸5动作延时 / 气缸5返回时间
TMR    T35 K20 K1
MPS
AND    T60	; 双夹耳气缸动作延时，气缸5动作延时
PLS    M692	; 继下
MPP
AND    T71	; 超神波焊接时间
AND    T60	; 双夹耳气缸动作延时，气缸5动作延时
AND    T35
MOV    K40 D1003	; 焊接流程
RST    M507	; 左超声波
RST    M514	; 右超声波
MOV    K4 D3003
LD     M692	; 继下
MOV    K1 D1004	; 主架子流程
LDP    T35
ZRST   M505 M506	; 右双夹 / 左双夹耳气缸
GROUPE
; K40 ???????
GROUP

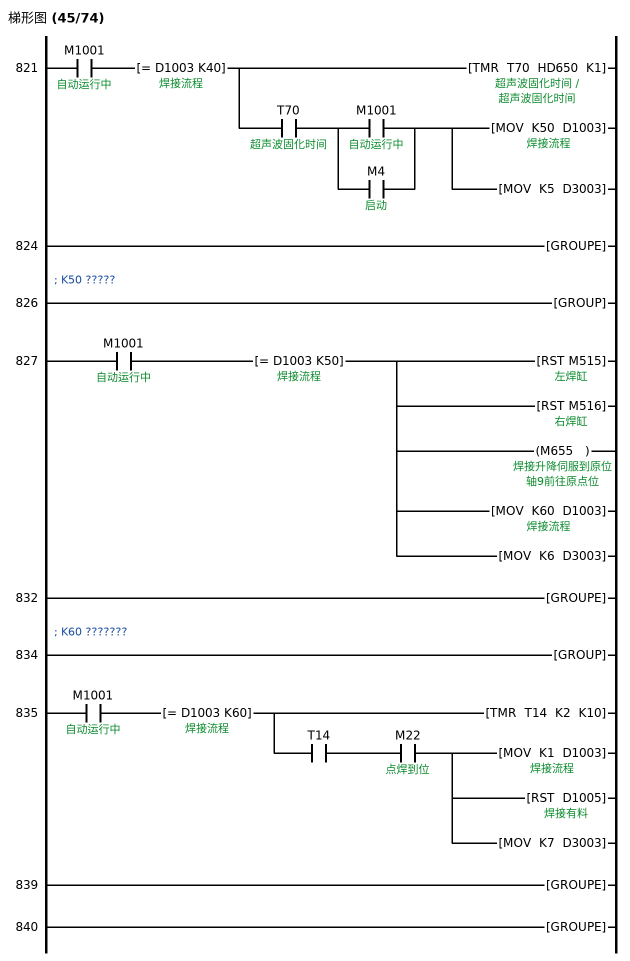
LD     M1001	; 自动运行中
AND=   D1003 K40	; 焊接流程
TMR    T70 HD650 K1	; 超声波固化时间 / 超声波固化时间
AND    T70	; 超声波固化时间
LD     M1001	; 自动运行中
OR     M4	; 启动
ANB
MOV    K50 D1003	; 焊接流程
MOV    K5 D3003
GROUPE
; K50 ?????
GROUP
LD     M1001	; 自动运行中
AND=   D1003 K50	; 焊接流程
RST    M515	; 左焊缸
RST    M516	; 右焊缸
OUT    M655	; 焊接升降伺服到原位 轴9前往原点位
MOV    K60 D1003	; 焊接流程
MOV    K6 D3003
GROUPE
; K60 ???????
GROUP
LD     M1001	; 自动运行中
AND=   D1003 K60	; 焊接流程
TMR    T14 K2 K10
AND    T14
AND    M22	; 点焊到位
MOV    K1 D1003	; 焊接流程
RST    D1005	; 焊接有料
MOV    K7 D3003
GROUPE
GROUPE

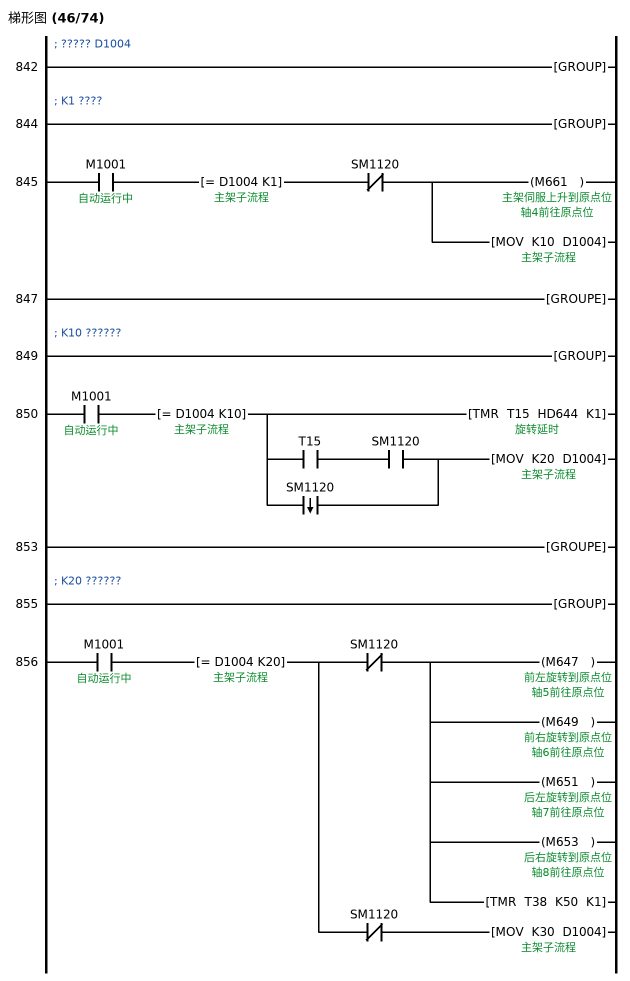
; ????? D1004
GROUP
; K1 ????
GROUP
LD     M1001	; 自动运行中
AND=   D1004 K1	; 主架子流程
ANI    SM1120
OUT    M661	; 主架伺服上升到原点位 轴4前往原点位
MOV    K10 D1004	; 主架子流程
GROUPE
; K10 ??????
GROUP
LD     M1001	; 自动运行中
AND=   D1004 K10	; 主架子流程
TMR    T15 HD644 K1	; 旋转延时
LD     T15
AND    SM1120
ORF    SM1120
ANB
MOV    K20 D1004	; 主架子流程
GROUPE
; K20 ??????
GROUP
LD     M1001	; 自动运行中
AND=   D1004 K20	; 主架子流程
MPS
ANI    SM1120
OUT    M647	; 前左旋转到原点位 轴5前往原点位
OUT    M649	; 前右旋转到原点位 轴6前往原点位
OUT    M651	; 后左旋转到原点位 轴7前往原点位
OUT    M653	; 后右旋转到原点位 轴8前往原点位
TMR    T38 K50 K1
MPP
ANI    SM1120
MOV    K30 D1004	; 主架子流程

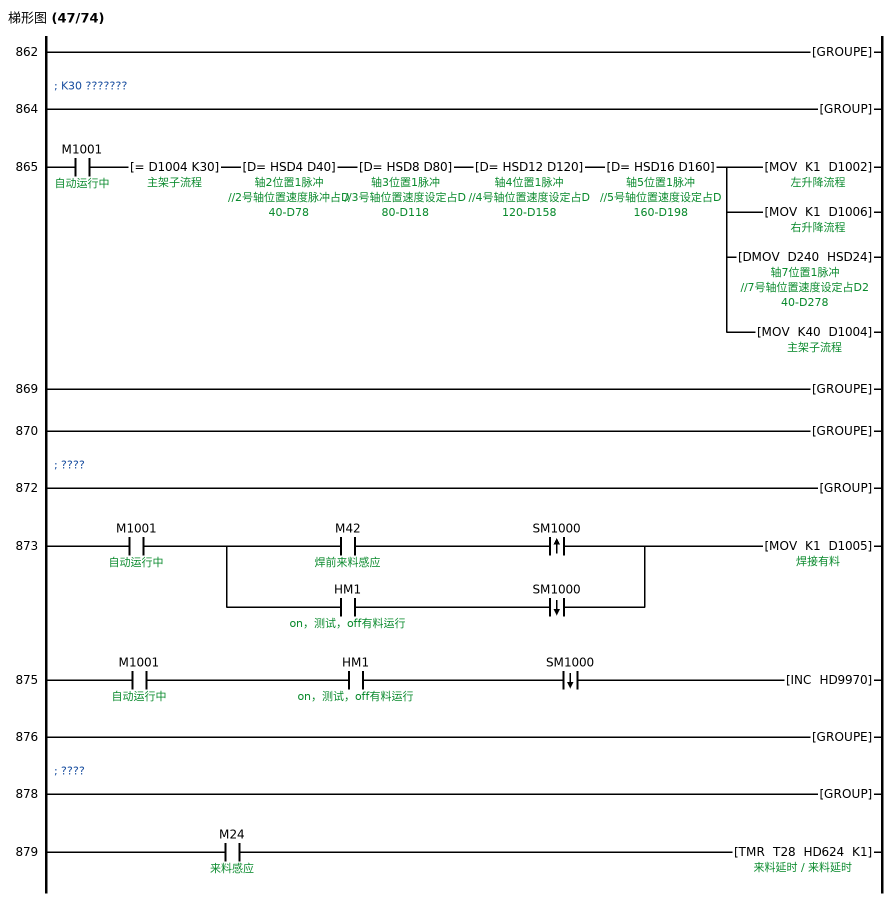
GROUPE
; K30 ???????
GROUP
LD     M1001	; 自动运行中
AND=   D1004 K30	; 主架子流程
DAND=  HSD4 D40	; 轴2位置1脉冲    //2号轴位置速度脉冲占D40-D78
DAND=  HSD8 D80	; 轴3位置1脉冲   //3号轴位置速度设定占D80-D118
DAND=  HSD12 D120	; 轴4位置1脉冲   //4号轴位置速度设定占D120-D158
DAND=  HSD16 D160	; 轴5位置1脉冲   //5号轴位置速度设定占D160-D198
MOV    K1 D1002	; 左升降流程
MOV    K1 D1006	; 右升降流程
DMOV   D240 HSD24	; 轴7位置1脉冲   //7号轴位置速度设定占D240-D278
MOV    K40 D1004	; 主架子流程
GROUPE
GROUPE
; ????
GROUP
LD     M1001	; 自动运行中
LD     M42	; 焊前来料感应
ANDP   SM1000
LD     HM1	; on，测试，off有料运行
ANDF   SM1000
ORB
ANB
MOV    K1 D1005	; 焊接有料
LD     M1001	; 自动运行中
AND    HM1	; on，测试，off有料运行
ANDF   SM1000
INC    HD9970
GROUPE
; ????
GROUP
LD     M24	; 来料感应
TMR    T28 HD624 K1	; 来料延时 / 来料延时

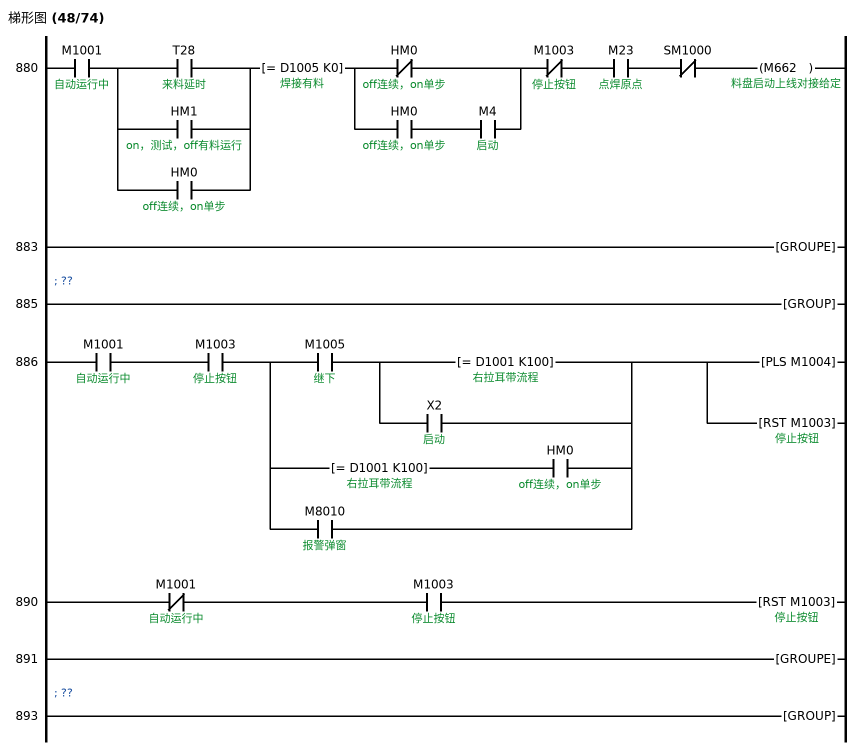
LD     M1001	; 自动运行中
LD     T28	; 来料延时
OR     HM1	; on，测试，off有料运行
OR     HM0	; off连续，on单步
ANB
AND=   D1005 K0	; 焊接有料
LDI    HM0	; off连续，on单步
LD     HM0	; off连续，on单步
AND    M4	; 启动
ORB
ANB
ANI    M1003	; 停止按钮
AND    M23	; 点焊原点
ANI    SM1000
OUT    M662	; 料盘启动上线对接给定
GROUPE
; ??
GROUP
LD     M1001	; 自动运行中
AND    M1003	; 停止按钮
LD     M1005	; 继下
LD=    D1001 K100	; 右拉耳带流程
OR     X2	; 启动
ANB
LD=    D1001 K100	; 右拉耳带流程
AND    HM0	; off连续，on单步
ORB
OR     M8010	; 报警弹窗
ANB
PLS    M1004
RST    M1003	; 停止按钮
LDI    M1001	; 自动运行中
AND    M1003	; 停止按钮
RST    M1003	; 停止按钮
GROUPE
; ??
GROUP

